(* PLC project Unnamed, Unknown Unnamed 1 *)
(* stored: creationDateTime 2025-06-20T22:38:36, modificationDateTime 2025-06-21T00:35:11 *)

PROGRAM comp
  VAR
    input1 AT %IX100.0 : BOOL;
    input2 AT %IX100.1 : BOOL;
    reset AT %IX100.2 : BOOL;
    load AT %IX100.3 : BOOL;
    output1 AT %QX100.0 : BOOL;
    output2 AT %QX100.1 : BOOL;
  END_VAR
  VAR
    R_TRIG0 : R_TRIG;
    R_TRIG1 : R_TRIG;
    CTU0 : CTU;
    CTU1 : CTU;
  END_VAR
  VAR  (* added by the conversion: wires and edge detectors of the diagram *)
    R_TRIG1_2 : R_TRIG;
    R_TRIG2 : R_TRIG;
  END_VAR

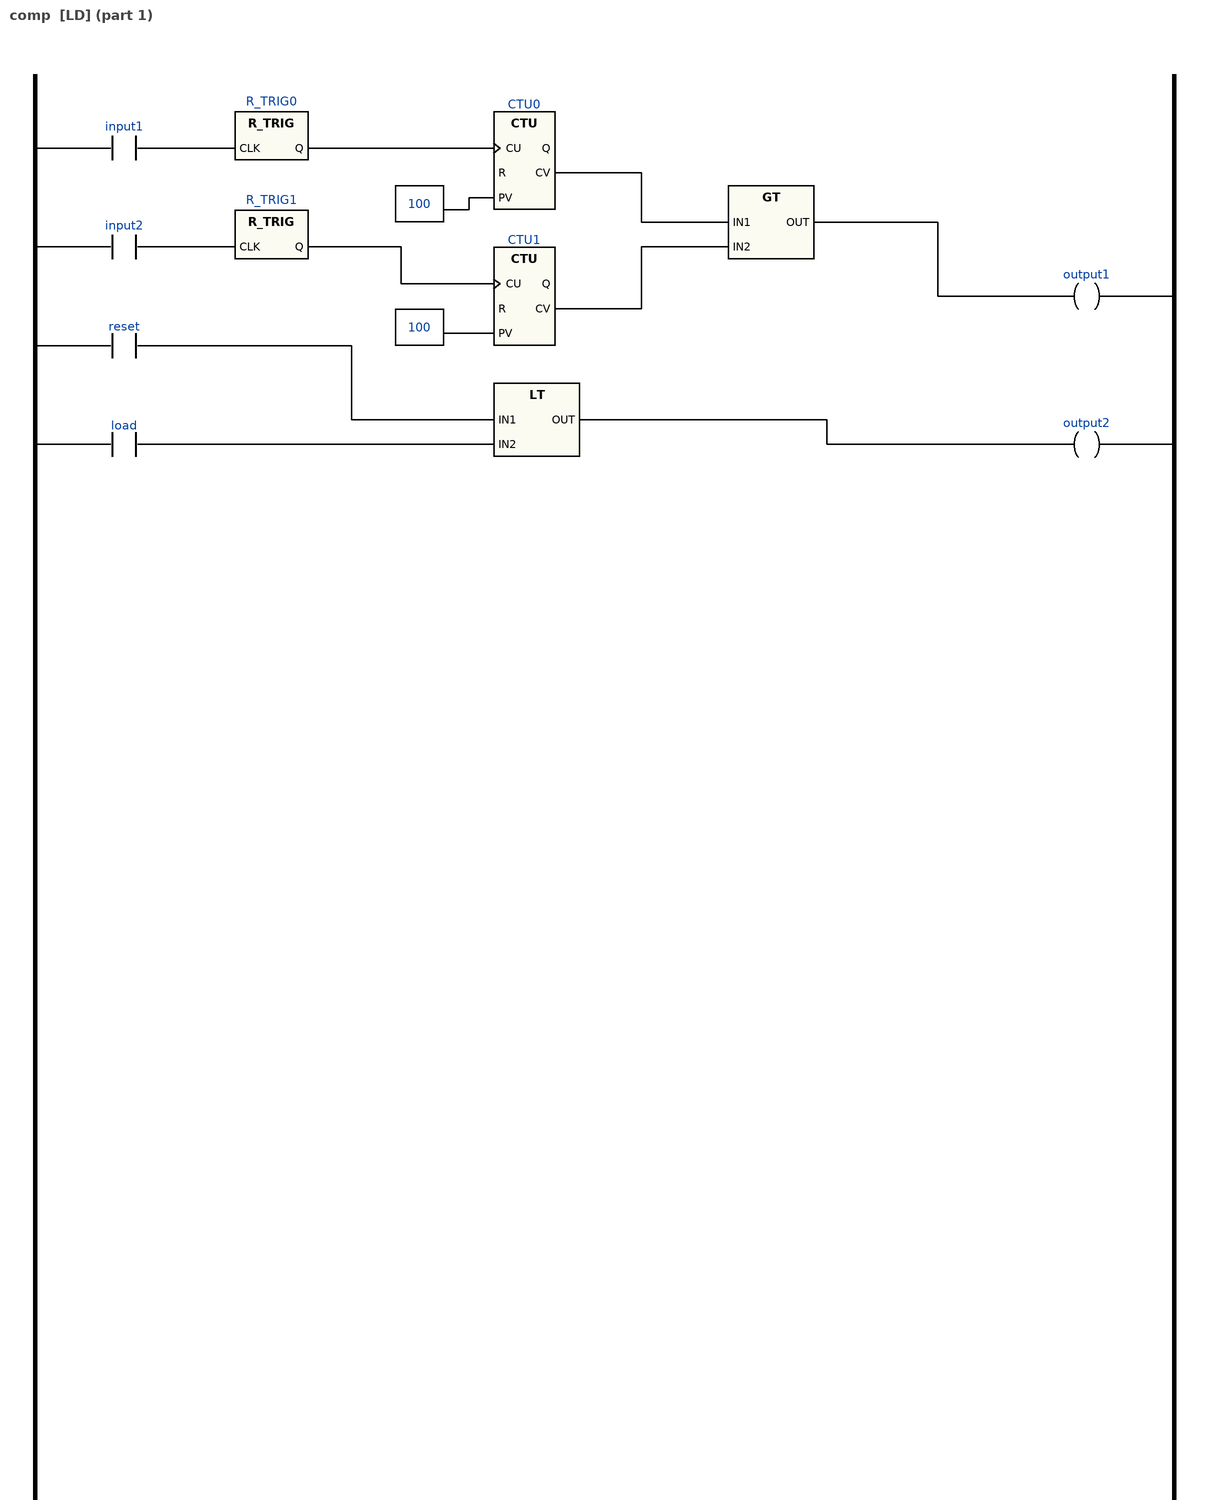
(* LD diagram, written out as Structured Text *)
R_TRIG0(CLK := input1);
R_TRIG1_2(CLK := R_TRIG0.Q);
CTU0(CU := R_TRIG1_2.Q, PV := 100);
R_TRIG1(CLK := input2);
R_TRIG2(CLK := R_TRIG1.Q);
CTU1(CU := R_TRIG2.Q, PV := 100);
output1 := CTU0.CV > CTU1.CV;
output2 := reset < load;
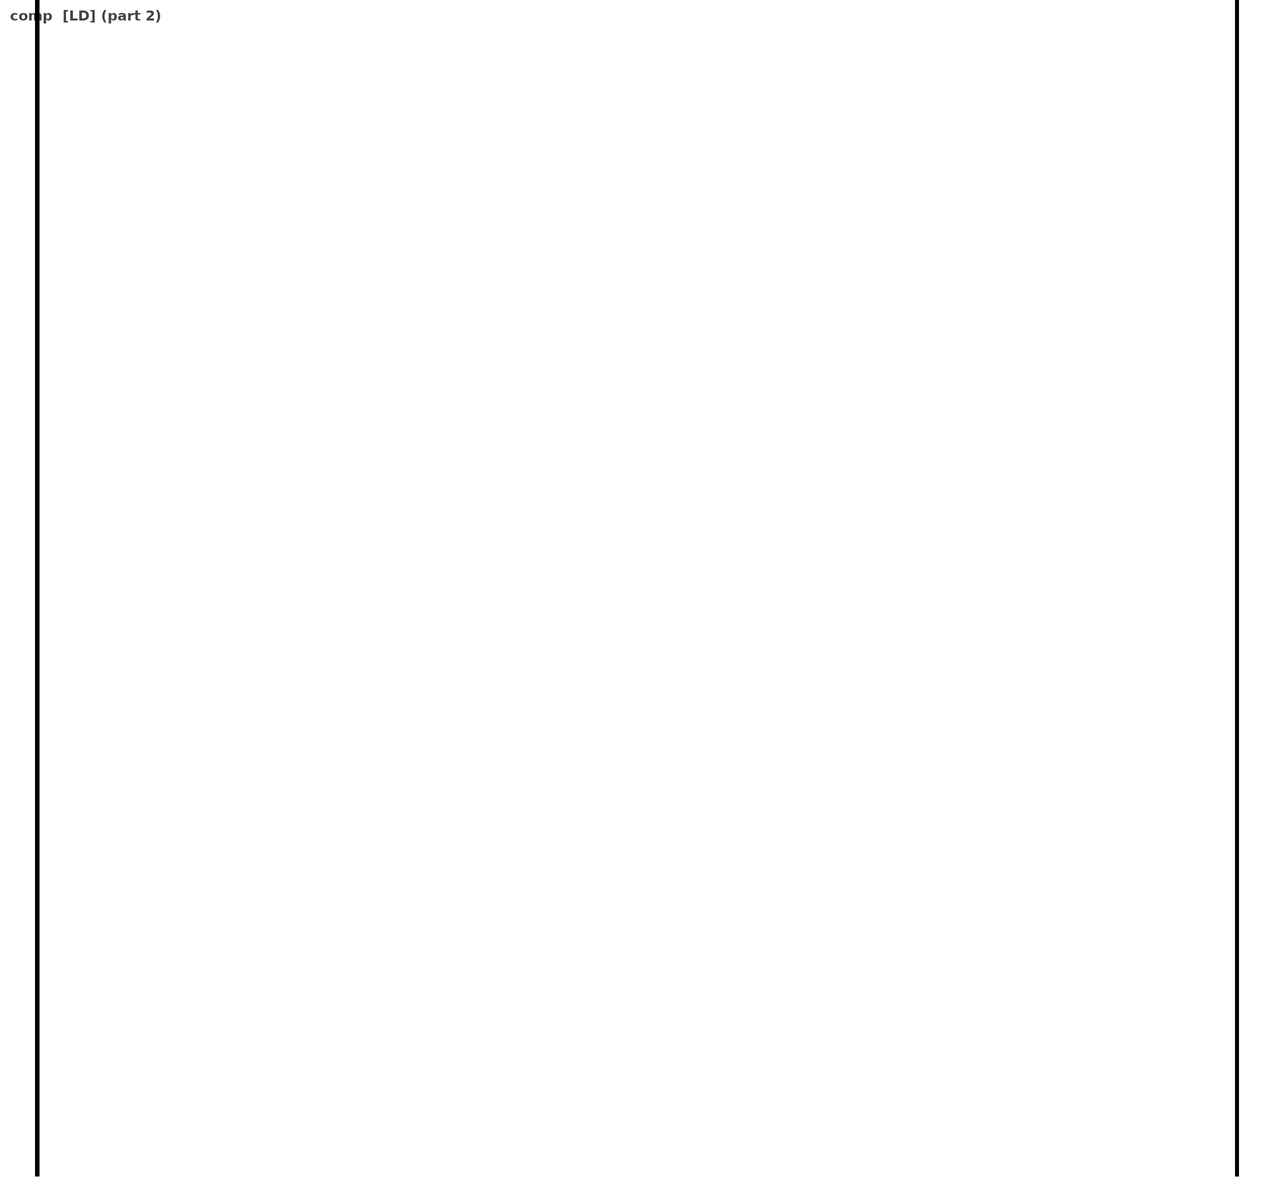
END_PROGRAM

CONFIGURATION Config0
  RESOURCE Res0 ON PLC
    TASK task0(INTERVAL := T#20ms, PRIORITY := 0);
    PROGRAM instance0 WITH task0 : comp;
  END_RESOURCE
END_CONFIGURATION
